Yaskawa INFORM job: PARK-POS-ZONE-3-AUTO.JBI

/JOB
//NAME PARK-POS-ZONE-3-AUTO
//POS
///NPOS 1,1,0,0,0,0
///TOOL 0
///POSTYPE PULSE
///PULSE
C00000=100644,-58707,-30728,-26719,55125,64105
BC00000=208121
//INST
///DATE 2018/10/01 15:23
///ATTR SC,RW
///GROUP1 RB1,BS1
NOP
MOVJ C00000 BC00000 VJ=20.00
END
